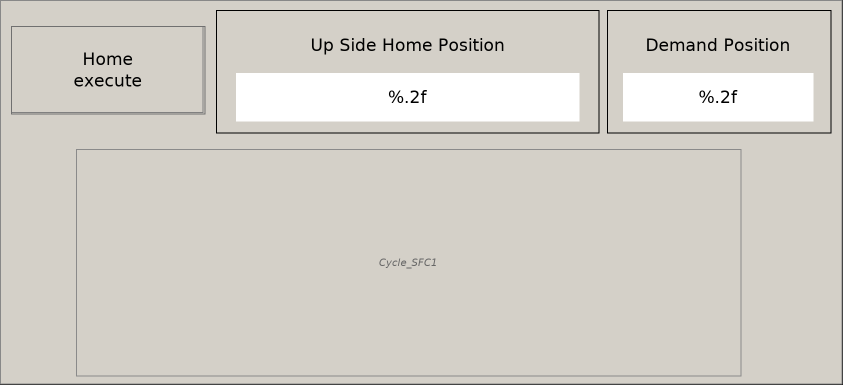
VISUALIZATION vHoming  // 843x385
VAR_IN_OUT
	fbHome:FB_DeadStopHomming;
END_VAR
    Rectangle (0,0 843x385)
    Button (11,26 194x88), "Home execute"
        toggle fbHome.bExecute
    Frame (76,149 665x227)
        shows Cycle_SFC1(fbCycle := fbHome.fb_SFC_Cycle)
    RoundedRectangle (607,10 224x123)
    Textfield (622,72 192x50), "%.2f", text variable: fbHome.iEndPosition
        OnMouseClick: write the text variable via Default
    Textfield (622,20 192x50), "Demand Position"
    RoundedRectangle (216,10 383x123)
    Textfield (235,20 346x50), "Up Side Home Position"
    Textfield (235,72 345x50), "%.2f", text variable: fbHome.fHomingPositionOffset
        OnMouseClick: write the text variable via Default
END_VISUALIZATION

(* stored: Version 1.1.0.1, ProductVersion 3.1.4024.11
   Visu vHoming: Id {32e6eb82-c4b1-4227-a456-de9833d928e6} *)
